{attribute 'qualified_only'}
{attribute 'strict'}
TYPE EFeedbackMsgPsdChuck :
(
	WaferPresenceMsg := 10
);
END_TYPE

(* stored: Version 1.1.0.1, ProductVersion 3.1.4024.12
   DUT EFeedbackMsgPsdChuck: Id {2e3b3e78-a67c-4499-88bc-cba3aecc8655} *)
